# EPICS substitutions: db/Beckhoff_3XXX/ecmcELM3602.substitutions
file "ecmc_analogInputArray-chX.template"
{
  pattern {CH_ID, DTYP,                FTVL    }
          {01,    "asynInt32ArrayIn",  "LONG" }
          {02,    "asynInt32ArrayIn",  "LONG" }
}

file "ecmcELM360X-stat-chX.template"
{
  pattern {CH_ID}
          {01   }
          {02   }
}

file "ecmc_controlWord-chX.template"
{
  pattern {CH_ID, KEY,   suffix,  sourceName, DESC             }
          {01,    "AI", "_Ctrl", "control",   "AI Control Word"}
          {02,    "AI", "_Ctrl", "control",   "AI Control Word"}
}
